FUNCTION_BLOCK CylControlILChanOL (* Composite Function Block Type *)
  (* Standard: 61499-2 *)
  (* Version 0.0, 7/14/2023, valeriy, nxtControl GmBH, template *)
  PACKAGE Main;
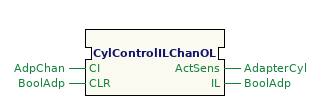
  SOCKETS
    CI : AdpChan;
    CLR : BoolAdp;
  END_SOCKETS
  PLUGS
    ActSens : AdapterCyl;
    IL : BoolAdp;
  END_PLUGS
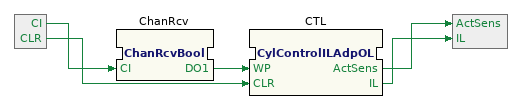
  FBS
    CTL : CylControlILAdpOL;
    ChanRcv : ChanRcvBool;
  END_FBS
  ADAPTER_CONNECTIONS
    ChanRcv.DO1 TO CTL.WP;
    CI TO ChanRcv.CI;
    CTL.ActSens TO ActSens;
    CLR TO CTL.CLR;
    CTL.IL TO IL;
  END_CONNECTIONS
END_FUNCTION_BLOCK
